(* IEC 61131-3 sources: Idecon_CheckWeigher_WP/plc_export, 11 files *)

(* ---- Idecon_BatchStats.st ---- *)
// ============================================================================
// DataType: Idecon_BatchStats
// Description: Statistiche batch da messaggio STATP (50 campi)
// Version: 1.0
// ============================================================================

TYPE Idecon_BatchStats :
STRUCT
    // === Header (Campi 1-7) ==================================================
    Timestamp               : STRING[32];       // Data/ora statistiche
    BatchStartTime          : STRING[32];       // Inizio batch
    ProductionOrder         : STRING[64];       // Ordine produzione
    ProductionCode          : STRING[64];       // Codice prodotto
    RecipeName              : STRING[32];       // Nome ricetta
    LineCode                : STRING[32];       // Codice linea
    SerialNumber            : STRING[16];       // Serial number

    // === Contatori Global Batch (Campi 8-22) =================================
    TotalProducts           : UDINT;            // Totale pezzi (Campo 8)
    TotalAccepted           : UDINT;            // Totale accettati (Campo 9)
    RejectedMinusMinus      : UDINT;            // Scartati -- (Campo 13)
    RejectedMinus           : UDINT;            // Scartati - (Campo 14)
    RejectedPlus            : UDINT;            // Scartati + (Campo 15)
    RejectedPlusPlus        : UDINT;            // Scartati ++ (Campo 16)
    CannotBeWeighed         : UDINT;            // Non pesabili (Campo 17)
    MetalDetected           : UDINT;            // Metallo rilevato (Campo 18)

    // === Metal Test (Campi 19-22) ============================================
    MetalTestsPerformed     : UDINT;            // Test metallo eseguiti
    MetalTestsPassed        : UDINT;            // Test superati
    MetalTestsFailed        : UDINT;            // Test falliti
    MetalTestsRefused       : UDINT;            // Test rifiutati

    // === Pesi Campione OK (Campi 10-12, 23-26) ===============================
    AverageWeight_g         : REAL;             // Peso medio accettati (g)
    MinWeight_g             : REAL;             // Peso minimo accettati (g)
    MaxWeight_g             : REAL;             // Peso massimo accettati (g)

    // Ultimo peso (Campi 23-26)
    LastWeightExact_g       : REAL;             // Ultimo peso esatto (g)
    LastWeightRounded_g     : REAL;             // Ultimo peso arrotondato (g)
    LastWeightDiff_g        : REAL;             // Ultimo delta (g)
    LastWeightClass         : STRING[16];       // Classe ultimo peso

    // === Contatori Incrementali (Campi 27-46) ================================
    IncrProducts            : UDINT;            // Incrementale totale
    IncrAccepted            : UDINT;            // Incrementale accettati
    IncrRejectedMM          : UDINT;            // Incrementale --
    IncrRejectedM           : UDINT;            // Incrementale -
    IncrRejectedP           : UDINT;            // Incrementale +
    IncrRejectedPP          : UDINT;            // Incrementale ++
    IncrCannotBeWeighed     : UDINT;            // Incrementale non pesabili
    IncrMetalDetected       : UDINT;            // Incrementale metallo

    // === KPI (Campi 47-50) ===================================================
    OKMinusProducts         : UDINT;            // OK- prodotti (Campo 48)
    OKMinusAccepted         : UDINT;            // OK- accettati (Campo 49)
    StandardDeviation_g     : REAL;             // Deviazione standard (Campo 50)

    // === KPI Calcolati =======================================================
    YieldPercentage         : REAL;             // Rendimento % (Accepted/Total*100)
    RejectionRate           : REAL;             // Tasso scarto %
    ProductionRate_PPM      : REAL;             // Pezzi al minuto
    TotalWeight_kg          : REAL;             // Peso totale kg

    // === Stato e Validità ====================================================
    BatchActive             : BOOL;             // Batch attivo
    DataValid               : BOOL;             // Dati validi
    ReceivedTime            : LINT;             // Timestamp ricezione
    LastUpdateTime          : LINT;             // Ultimo aggiornamento
    ParseError              : BOOL;             // Errore parsing
    ErrorCode               : UINT;             // Codice errore

    // === Campi Extra dal Batch ===============================================
    ExtraField1             : STRING[64];       // Campo extra 1
    ExtraField2             : STRING[64];       // Campo extra 2
    UserName                : STRING[32];       // Nome operatore

END_STRUCT;
END_TYPE

(* ---- Idecon_Command.st ---- *)
// ============================================================================
// DataType: Idecon_Command
// Description: Struttura per gestione comando singolo verso bilancia
// ============================================================================

TYPE Idecon_Command :
STRUCT
    // === Input (da programma chiamante) ======================================
    Execute                 : BOOL;             // Esegui comando (fronte salita)
    Command                 : STRING[255];      // Stringa comando (es. "STATSV")
    Timeout                 : TIME := T#5S;     // Timeout attesa risposta

    // === Output (da FB_IDECON_Client) ========================================
    Done                    : BOOL;             // Comando completato con successo
    Busy                    : BOOL;             // Comando in esecuzione
    Error                   : BOOL;             // Errore durante esecuzione
    ErrorID                 : WORD;             // Codice errore specifico

    // === Risposta ============================================================
    Response                : STRING[512];      // Risposta testuale da bilancia
    ResponseRaw             : ARRAY[0..511] OF BYTE;  // Risposta come array byte
    ResponseLen             : UINT;             // Lunghezza risposta in bytes
    ResponseTime_ms         : UDINT;            // Tempo risposta (ms)

    // === Timestamp ===========================================================
    ExecuteTime             : LINT;             // Quando è stato eseguito
    DoneTime                : LINT;             // Quando è stato completato

END_STRUCT;
END_TYPE

(* ---- Idecon_CommStatus.st ---- *)
// ============================================================================
// DataType: Idecon_CommStatus
// Description: Stato comunicazione TCP con bilancia IDECON
// ============================================================================

TYPE Idecon_CommStatus :
STRUCT
    // === Stato Connessione ===================================================
    Connected               : BOOL;             // Socket connesso fisicamente
    Online                  : BOOL;             // Comunicazione attiva (ultimo msg < timeout)
    Ready                   : BOOL;             // Pronto per inviare comandi

    // === Statistiche Comunicazione ===========================================
    RxCount                 : UDINT;            // Totale messaggi ricevuti
    TxCount                 : UDINT;            // Totale comandi inviati
    ErrorCount              : UDINT;            // Contatore errori
    RetryCount              : UINT;             // Retry in corso

    // === Timestamp ===========================================================
    LastRxTime              : LINT;             // Timestamp ultimo messaggio ricevuto (Unix ms)
    LastTxTime              : LINT;             // Timestamp ultimo comando inviato
    ConnectionTime          : LINT;             // Timestamp connessione stabilita

    // === Errori ==============================================================
    LastError               : WORD;             // Codice ultimo errore
    LastErrorTime           : LINT;             // Timestamp ultimo errore

    // === Stato Dettagliato ===================================================
    StatusCode              : STRING[8];        // Ultimo STATSV ricevuto
    WorkMode                : UINT;             // 1=LOCAL, 2=REMOTE, 3=MAINTENANCE
    IsLocalMode             : BOOL;             // TRUE se in LOCAL
    IsRemoteMode            : BOOL;             // TRUE se in REMOTE

END_STRUCT;
END_TYPE

(* ---- Idecon_Config.st ---- *)
// ============================================================================
// DataType: Ideon_Config
// Description: Configurazione rete e parametri bilancia IDECON
// ============================================================================

TYPE Idecon_Config :
STRUCT
    // === Parametri Rete ======================================================
    IpAddress               : STRING[15] := '172.16.224.210';  // IP bilancia
    TcpPort                 : UINT := 50000;                    // Porta TCP

    // === Timeout (millisecondi) ==============================================
    ConnectionTimeout_ms    : UDINT := 10000;                   // Timeout connessione
    CommandTimeout_ms       : UDINT := 5000;                    // Timeout comando
    ResponseTimeout_ms      : UDINT := 5000;                    // Timeout risposta

    // === Polling =============================================================
    PollInterval_ms         : UDINT := 5000;                    // Intervallo polling STATSV

    // === Retry ===============================================================
    MaxRetries              : UINT := 3;                        // Numero max retry

    // === MSGFILTER ===========================================================
    MsgFilterValue          : UINT := 23;                       // 0b10111 = risp+err+ev+pesi

    // === Statistiche =========================================================
    StatsCadency_sec        : UINT := 30;                       // Frequenza STATP (secondi)

    // === Abilitazione ========================================================
    Connect                 : BOOL := FALSE;                    // Abilita connessione
    AutoReconnect           : BOOL := TRUE;                     // Riconnessione automatica

END_STRUCT;
END_TYPE

(* ---- Idecon_LocalStats.st ---- *)
// ============================================================================
// DataType: Idecon_LocalStats
// Description: Statistiche locali calcolate dal PLC (indipendenti da bilancia)
// ============================================================================

TYPE Idecon_LocalStats :
STRUCT
    // === Contatori Totali ====================================================
    TotalWeights            : UDINT;            // Totale pesi ricevuti
    TotalAccepted           : UDINT;            // Totale OK
    TotalRejected           : UDINT;            // Totale scartati
    TotalExpelled           : UDINT;            // Totale espulsi

    // === Contatori per Categoria =============================================
    CountOK                 : UDINT;            // Solo OK
    CountOKPlus             : UDINT;            // OK+
    CountOKMinus            : UDINT;            // OK-
    CountPlus               : UDINT;            // +
    CountPlusPlus           : UDINT;            // ++
    CountMinus              : UDINT;            // -
    CountMinusMinus         : UDINT;            // --
    CountMetal              : UDINT;            // Con metallo

    // === Pesi (calcolati in g) ===============================================
    SumWeight_g             : REAL;             // Somma pesi (per media)
    AvgWeight_g             : REAL;             // Media pesi
    MinWeight_g             : REAL;             // Peso minimo rilevato
    MaxWeight_g             : REAL;             // Peso massimo rilevato

    // === Timing ==============================================================
    FirstWeightTime         : LINT;             // Timestamp prima pesata
    LastWeightTime          : LINT;            // Timestamp ultima pesata
    ProductionTime_sec      : UDINT;            // Tempo produzione (secondi)

    // === Allarmi =============================================================
    Error30_Count           : UDINT;            // Quanti errori 30 ricevuti
    OtherErrors_Count       : UDINT;            // Altri errori

    // === Reset ===============================================================
    Reset                   : BOOL;             // Azzera contatori

END_STRUCT;
END_TYPE

(* ---- Idecon_Types.st ---- *)
// ============================================================================
// DataType: Idecon_Status
// Description: Stato macchina da risposta STATSV
// Version: 1.0
// ============================================================================

TYPE Idecon_Status :
STRUCT
    // === Codice Stato (8 caratteri) ==========================================
    StatusCode              : STRING[8];        // Codice completo (es. "20110011")

    // === Posizione 1: Stato Motori ==========================================
    MotorStatus             : UINT;             // 0=Fermo, 1=Regolazione, 2=Pronto, 3=Standby, 4=Ripresa
    MotorRunning            : BOOL;             // TRUE se in moto

    // === Posizione 2: Produzione =============================================
    ProductionStarted       : BOOL;             // 1=Produzione attiva

    // === Posizione 3-5: Allarmi ==============================================
    HasErrors               : BOOL;             // 1=Errori presenti
    HasWarnings             : BOOL;             // 1=Warning presenti
    HasMessages             : BOOL;             // 1=Messaggi presenti

    // === Posizione 6: Statistiche ============================================
    StatsEnabled            : BOOL;             // 1=Invio STATP abilitato

    // === Posizione 7: Modalità Operativa =====================================
    WorkMode                : UINT;             // 1=LOCAL, 2=REMOTE, 3=MAINTENANCE
    IsLocalMode             : BOOL;             // TRUE se in LOCAL
    IsRemoteMode            : BOOL;             // TRUE se in REMOTE
    IsMaintenanceMode       : BOOL;             // TRUE se in MAINTENANCE

    // === Posizione 8: Connessione ============================================
    ConnectionStatus        : UINT;             // Stato connessione

    // === Timestamp ===========================================================
    ReceivedTime            : LINT;             // Timestamp ricezione
    Valid                   : BOOL;             // Dati validi

END_STRUCT;
END_TYPE

// ============================================================================
// DataType: Idecon_EventData
// Description: Dati evento da messaggio EVENT
// Version: 1.0
// ============================================================================

TYPE Idecon_EventData :
STRUCT
    Timestamp               : STRING[32];       // Data/ora evento
    ProductionOrder         : STRING[64];       // Ordine
    BatchCode               : STRING[64];       // Batch
    RecipeName              : STRING[32];       // Ricetta
    LineCode                : STRING[32];       // Linea
    SerialNumber            : STRING[16];       // Serial

    EventCode               : UINT;             // Codice evento (1000-9999)
    EventDescription        : STRING[255];      // Descrizione testuale
    Operator                : STRING[32];       // Operatore

    // Flag comuni
    IsError                 : BOOL;             // TRUE se errore
    IsWarning               : BOOL;             // TRUE se warning
    IsInfo                  : BOOL;             // TRUE se informativo

    // Timestamp
    ReceivedTime            : LINT;
    Valid                   : BOOL;

END_STRUCT;
END_TYPE

// ============================================================================
// DataType: Idecon_Config
// Description: Configurazione connessione IDECON
// Version: 1.0
// ============================================================================

TYPE Idecon_Config :
STRUCT
    // === Parametri Rete ======================================================
    IpAddress               : STRING[15];       // IP bilancia (es. "172.16.224.210")
    TcpPort                 : UINT;             // Porta (default 50000)

    // === Timeout =============================================================
    ConnectionTimeout_ms    : UDINT;            // Timeout connessione (ms)
    CommandTimeout_ms       : UDINT;            // Timeout comando (ms)
    ResponseTimeout_ms      : UDINT;            // Timeout risposta (ms)

    // === Polling =============================================================
    PollInterval_ms         : UDINT;            // Intervallo polling STATSV (ms)

    // === Retry ===============================================================
    MaxRetries              : UINT;             // Numero massimo retry

    // === MSGFILTER ===========================================================
    MsgFilterValue          : UINT;             // Valore MSGFILTER (default 23)

    // === Statistiche =========================================================
    StatsCadency_sec        : UINT;             // Frequenza STATP (default 30s)

    // === Abilitazione ========================================================
    Connect                 : BOOL;             // Abilita connessione
    AutoReconnect           : BOOL;             // Riconnessione automatica

END_STRUCT;
END_TYPE

(* ---- Idecon_WeightData.st ---- *)
// ============================================================================
// DataType: Idecon_WeightData
// Description: Struttura dati per messaggio WEIGHT dalla bilancia IDECON
// Version: 1.0
// ============================================================================

TYPE Idecon_WeightData :
STRUCT
    // === Identificazione =====================================================
    Timestamp               : STRING[32];       // Data/ora pesata (yyyy.mm.dd hh:mm:ss:msec)
    ProductionOrder         : STRING[64];       // Ordine produzione
    BatchCode               : STRING[64];       // Codice batch/lotto
    RecipeName              : STRING[32];       // Nome ricetta (es. "225g")
    LineCode                : STRING[32];       // Codice linea
    SerialNumber            : STRING[16];       // Serial number bilancia

    // === Valori numerici (in milligrammi) ====================================
    WeightMg                : DINT;             // Peso rilevato in mg
    DeltaMg                 : DINT;             // Delta da peso nominale in mg
    Classification          : UDINT;            // Bitmap classificazione (19 bit)

    // === Flag decodificati (19 bit di Classification) ========================
    // Bit 0-2: Caratteristiche fisiche
    FlagProductTooLong      : BOOL;             // Prodotto troppo lungo (Bit 0)
    FlagProductTooShort     : BOOL;             // Prodotto troppo corto (Bit 1)
    FlagMetal               : BOOL;             // Rilevato metallo (Bit 2)

    // Bit 3-7: Categorie peso
    FlagWeightPlusPlus      : BOOL;             // Categoria ++ (Bit 3)
    FlagWeightPlus          : BOOL;             // Categoria + (Bit 4)
    FlagWeightMinusMinus    : BOOL;             // Categoria -- (Bit 5)
    FlagWeightMinus         : BOOL;             // Categoria - (Bit 6)
    FlagWeightOK            : BOOL;             // Categoria OK (Bit 7)

    // Bit 8-11: Condizioni speciali
    FlagExpelled            : BOOL;             // Espulso (Bit 8)
    FlagProductTooClose     : BOOL;             // Prodotto troppo vicino (Bit 9)
    FlagNewDynamicTare      : BOOL;             // Nuova tara dinamica (Bit 10)
    FlagIncorrectTare       : BOOL;             // Tara incorretta (Bit 11)

    // Bit 12-13: Fuori range
    FlagAboveMaxCapacity    : BOOL;             // Sopra capacità max (Bit 12)
    FlagBelowMinCapacity    : BOOL;             // Sotto capacità min (Bit 13)

    // Bit 14-18: Condizioni OK speciali
    FlagOKMinusAccepted     : BOOL;             // OK- accettato (Bit 14)
    FlagNoUpstreamConsent   : BOOL;             // No consenso upstream (Bit 15)
    FlagInvalidPreweight    : BOOL;             // Peso pre-pesata invalido (Bit 16)
    FlagOKAboveNominal      : BOOL;             // OK sopra nominale (Bit 17)
    FlagOKBelowNominal      : BOOL;             // OK sotto nominale (Bit 18)

    // === Validità e timestamp ================================================
    Valid                   : BOOL;             // Dati validi (ricevuti e parsati)
    ReceivedTime            : LINT;             // Timestamp ricezione (Unix ms)
    ParseError              : BOOL;             // Errore parsing
    ErrorCode               : UINT;             // Codice errore parsing

END_STRUCT;
END_TYPE

(* ---- IdeconInterface.st ---- *)
// ============================================================================
// DataType: IdeconInterface
// Description: Struttura principale unificata per gestione bilancia IDECON
//              Unica variabile in Global Variables: G_Idecon : IdeconInterface
// Version: 1.0
// ============================================================================

TYPE IdeconInterface :
STRUCT
    // === CONFIGURAZIONE (inizializzata in HSM_SpecificationsSetting) ========
    // Esempio: G_Idecon.Config.IpAddress := '172.16.224.210';
    Config                  : Idecon_Config;

    // === SOCKET TCP (gestito da FB_IDECON_Client) ===========================
    // Non modificare direttamente, usare FB
    Socket                  : _sSOCKET;

    // === STATO COMUNICAZIONE =================================================
    // Monitoraggio stato connessione e online/offline
    Comm                    : Idecon_CommStatus;

    // === DATI RICEVUTI DALLA BILANCIA ========================================
    // Ultimi dati aggiornati automaticamente
    LastWeight              : Idecon_WeightData;    // Ultima pesata WEIGHT
    BatchStats              : Idecon_BatchStats;    // Statistiche STATP
    Status                  : Idecon_Status;        // Stato macchina STATSV
    LastEvent               : Idecon_EventData;     // Ultimo evento EVENT

    // === COMANDO ATTIVO ======================================================
    // Per inviare comandi alla bilancia
    Cmd                     : Idecon_Command;

    // === STATISTICHE LOCALI PLC ==============================================
    // Contatori e calcoli fatti dal PLC
    Stats                   : Idecon_LocalStats;

    // === FLAG ERRORE SISTEMA =================================================
    // TRUE quando c'è errore grave comunicazione
    SystemError             : BOOL;

    // === VERSIONE E DIAGNOSTICA ==============================================
    Version                 : UINT := 100;          // Versione struct (1.00)

END_STRUCT;
END_TYPE

(* ---- IDECON_Utils.st ---- *)
// ============================================================================
// Function: IDECON_StartsWith
// Description: Verifica se una stringa inizia con un prefisso
// ============================================================================

FUNCTION IDECON_StartsWith : BOOL
VAR_INPUT
    Str                     : STRING[512];      // Stringa da verificare
    Prefix                  : STRING[64];       // Prefisso da cercare
END_VAR

VAR
    StrLen                  : UINT;
    PrefixLen               : UINT;
END_VAR;

StrLen := LEN(Str);
PrefixLen := LEN(Prefix);

IF PrefixLen = 0 THEN
    IDECON_StartsWith := TRUE;
    RETURN;
END_IF;

IF StrLen < PrefixLen THEN
    IDECON_StartsWith := FALSE;
    RETURN;
END_IF;

IDECON_StartsWith := (LEFT(Str, PrefixLen) = Prefix);

END_FUNCTION

// ============================================================================
// Function: IDECON_FieldAt
// Description: Estrae campo N da stringa delimitata
// ============================================================================

FUNCTION IDECON_FieldAt : STRING[64]
VAR_INPUT
    Str                     : STRING[512];      // Stringa sorgente
    FieldNum                : UINT;             // Numero campo (1-based)
    Delimiter               : STRING[1];        // Delimitatore
END_VAR

VAR
    i                       : INT;
    CurrentField            : UINT;
    StartPos                : INT;
    StrLen                  : UINT;
END_VAR;

StrLen := LEN(Str);
IF StrLen = 0 OR FieldNum = 0 THEN
    IDECON_FieldAt := '';
    RETURN;
END_IF;

CurrentField := 1;
StartPos := 1;

FOR i := 1 TO INT#(StrLen) DO
    IF MID(Str, 1, UINT#(i)) = Delimiter THEN
        IF CurrentField = FieldNum THEN
            // Campo trovato
            IDECON_FieldAt := MID(Str, UINT#(i - StartPos), UINT#(StartPos));
            RETURN;
        END_IF;
        CurrentField := CurrentField + 1;
        StartPos := i + 1;
    END_IF;
END_FOR;

// Ultimo campo
IF CurrentField = FieldNum THEN
    IDECON_FieldAt := MID(Str, UINT#(StrLen - StartPos + 1), UINT#(StartPos));
ELSE
    IDECON_FieldAt := '';
END_IF;

END_FUNCTION

// ============================================================================
// Function: IDECON_ParseHexDword
// Description: Converte stringa esadecimale in UDINT
// ============================================================================

FUNCTION IDECON_ParseHexDword : UDINT
VAR_INPUT
    HexStr                  : STRING[16];       // Stringa hex (es. "20480")
END_VAR

VAR
    Result                  : UDINT;
    i                       : INT;
    StrLen                  : UINT;
    Digit                   : BYTE;
    CharVal                 : UDINT;
END_VAR;

StrLen := LEN(HexStr);
Result := UDINT#0;

FOR i := 1 TO INT#(StrLen) DO
    Digit := STRING_TO_BYTE(MID(HexStr, 1, UINT#(i)));

    IF Digit >= BYTE#48 AND Digit <= BYTE#57 THEN
        // '0'-'9'
        CharVal := BYTE_TO_UDINT(Digit) - UDINT#48;
    ELSIF Digit >= BYTE#65 AND Digit <= BYTE#70 THEN
        // 'A'-'F'
        CharVal := BYTE_TO_UDINT(Digit) - UDINT#55;
    ELSIF Digit >= BYTE#97 AND Digit <= BYTE#102 THEN
        // 'a'-'f'
        CharVal := BYTE_TO_UDINT(Digit) - UDINT#87;
    ELSE
        CONTINUE; // Carattere non valido, salta
    END_IF;

    Result := Result * UDINT#16 + CharVal;
END_FOR;

IDECON_ParseHexDword := Result;

END_FUNCTION

(* ---- FB_IDECON_Client.st ---- *)
// ============================================================================
// Function Block: FB_IDECON_Client
// Description: Client TCP per comunicazione con bilancia IDECON
// Version: 1.0
// ============================================================================

FUNCTION_BLOCK FB_IDECON_Client
VAR_INPUT
    Execute                 : BOOL;             // Esegui comando
    Command                 : STRING[255];      // Comando da inviare
    Timeout                 : TIME := T#5S;     // Timeout risposta
END_VAR

VAR_OUTPUT
    Done                    : BOOL;             // Comando completato con successo
    Busy                    : BOOL;             // In esecuzione
    Error                   : BOOL;             // Errore
    ErrorID                 : WORD;             // Codice errore (0=nessuno)
    Response                : STRING[512];      // Risposta ricevuta
    ResponseRaw             : ARRAY[0..511] OF BYTE; // Risposta raw bytes
    ResponseLen             : UINT;             // Lunghezza risposta
END_VAR

VAR_IN_OUT
    Socket                  : _sSOCKET;         // Socket TCP
END_VAR

VAR
    // Stato FSM
    State                   : INT := 0;         // Stato macchina

    // Timer
    TimeoutTimer            : TON;              // Timer timeout
    RetryTimer              : TON;              // Timer retry

    // Buffer
    SendBuffer              : ARRAY[0..511] OF BYTE;
    RecvBuffer              : ARRAY[0..1023] OF BYTE;
    CmdLen                  : UINT;
    RetryCount              : INT := 0;
    MaxRetries              : INT := 3;

    // Costanti protocollo
    STX                     : BYTE := BYTE#16#02;  // Start of Text
    ETX                     : BYTE := BYTE#16#03;  // End of Text

    // Variabili interne
    i                       : INT;
    j                       : INT;
    StrLen                  : UINT;
    RecvDone                : BOOL;
    SendDone                : BOOL;

END_VAR

// Stati FSM
// 0: Idle
// 1: Prepara comando
// 2: Invia STX
// 3: Invia comando
// 4: Invia ETX
// 5: Attendi risposta
// 6: Ricevi dati
// 7: Parsa risposta
// 8: Completato
// 9: Errore

// ============================================================================
// IMPLEMENTAZIONE
// ============================================================================

IF NOT Execute AND State <> 0 THEN
    // Reset su fronte negativo Execute
    State := 0;
    Busy := FALSE;
END_IF;

CASE State OF

    0: // Idle
        Done := FALSE;
        Error := FALSE;
        ErrorID := WORD#0;
        Busy := FALSE;
        RetryCount := 0;

        IF Execute THEN
            State := 1;
            Busy := TRUE;
        END_IF;

    1: // Prepara comando
        // Prepara buffer: STX + Comando + ETX
        StrLen := LEN(Command);

        IF StrLen = 0 OR StrLen > 250 THEN
            Error := TRUE;
            ErrorID := WORD#1; // Comando vuoto o troppo lungo
            State := 9;
        ELSE
            // Copia comando in buffer
            FOR i := 0 TO INT#(StrLen - 1) DO
                SendBuffer[i + 1] := STRING_TO_BYTE(MID(Command, 1, UINT#(i + 1)));
            END_FOR;

            CmdLen := StrLen;
            State := 2;
        END_IF;

    2: // Invia STX
        Socket.Send(ADR(STX), 1);

        IF Socket.Done THEN
            State := 3;
        ELSIF Socket.Error THEN
            Error := TRUE;
            ErrorID := Socket.ErrorID;
            State := 9;
        END_IF;

    3: // Invia comando
        Socket.Send(ADR(SendBuffer[1]), CmdLen);

        IF Socket.Done THEN
            State := 4;
        ELSIF Socket.Error THEN
            Error := TRUE;
            ErrorID := Socket.ErrorID;
            State := 9;
        END_IF;

    4: // Invia ETX
        Socket.Send(ADR(ETX), 1);

        IF Socket.Done THEN
            State := 5;
            TimeoutTimer(IN := TRUE, PT := Timeout);
        ELSIF Socket.Error THEN
            Error := TRUE;
            ErrorID := Socket.ErrorID;
            State := 9;
        END_IF;

    5: // Attendi risposta
        TimeoutTimer(IN := TRUE);

        IF TimeoutTimer.Q THEN
            // Timeout - retry?
            IF RetryCount < MaxRetries THEN
                RetryCount := RetryCount + 1;
                State := 1; // Riprova
                TimeoutTimer(IN := FALSE);
            ELSE
                Error := TRUE;
                ErrorID := WORD#16#8001; // Timeout
                State := 9;
            END_IF;
        END_IF;

        // Controlla se ci sono dati
        IF Socket.Available > 0 THEN
            State := 6;
            TimeoutTimer(IN := FALSE);
        END_IF;

    6: // Ricevi dati
        Socket.Recv(ADR(RecvBuffer), SIZEOF(RecvBuffer), RecvLen);

        IF Socket.Done THEN
            State := 7;
        ELSIF Socket.Error THEN
            Error := TRUE;
            ErrorID := Socket.ErrorID;
            State := 9;
        END_IF;

    7: // Parsa risposta
        // Rimuovi STX e ETX se presenti
        IF RecvLen > 0 THEN
            j := 0;
            FOR i := 0 TO INT#(RecvLen - 1) DO
                // Salta STX iniziale
                IF i = 0 AND RecvBuffer[i] = STX THEN
                    CONTINUE;
                END_IF;
                // Salta ETX finale
                IF i = INT#(RecvLen - 1) AND RecvBuffer[i] = ETX THEN
                    CONTINUE;
                END_IF;
                // Copia byte valido
                ResponseRaw[j] := RecvBuffer[i];
                j := j + 1;
            END_FOR;

            // Converti in stringa
            Response := '';
            FOR i := 0 TO j - 1 DO
                IF ResponseRaw[i] >= BYTE#32 AND ResponseRaw[i] <= BYTE#126 THEN
                    Response := CONCAT(Response, BYTE_TO_STRING(ResponseRaw[i]));
                END_IF;
            END_FOR;

            ResponseLen := UINT#(j);
        END_IF;

        State := 8;

    8: // Completato
        Done := TRUE;
        Busy := FALSE;
        Error := FALSE;

        IF NOT Execute THEN
            State := 0;
        END_IF;

    9: // Errore
        Error := TRUE;
        Busy := FALSE;
        Done := FALSE;

        IF NOT Execute THEN
            State := 0;
        END_IF;

END_CASE;

END_FUNCTION_BLOCK

(* ---- FB_ParseWeightMessage.st ---- *)
// ============================================================================
// Function Block: FB_ParseWeightMessage
// Description: Parsa messaggio WEIGHT dalla bilancia IDECON
// Version: 1.0
// ============================================================================

FUNCTION_BLOCK FB_ParseWeightMessage
VAR_INPUT
    Enable                  : BOOL;             // Abilita parsing
    Message                 : STRING[512];      // Messaggio da parsare
    MessageRaw              : ARRAY[0..511] OF BYTE;
    MessageLen              : UINT;
END_VAR

VAR_OUTPUT
    Done                    : BOOL;             // Parsing completato
    Error                   : BOOL;             // Errore parsing
    ErrorCode               : UINT;             // Codice errore
    WeightData              : Idecon_WeightData; // Dati peso parsati
END_VAR

VAR
    // Variabili interne
    MsgTemp                 : STRING[512];
    Parts                   : ARRAY[0..10] OF STRING[64];
    NumParts                : INT;
    i                       : INT;
    Pos                     : INT;
    LastPos                 : INT;
    ClassificationValue     : UDINT;

END_VAR

// ============================================================================
// IMPLEMENTAZIONE
// ============================================================================

IF NOT Enable THEN
    Done := FALSE;
    Error := FALSE;
    ErrorCode := UINT#0;
    RETURN;
END_IF;

// Verifica prefisso WEIGHT=
IF NOT IDECON_StartsWith(Message, 'WEIGHT=') THEN
    Error := TRUE;
    ErrorCode := UINT#1; // Prefisso non valido
    RETURN;
END_IF;

// Rimuovi prefisso
MsgTemp := DELETE(Message, 7, 1); // Rimuovi "WEIGHT="

// Split per |
NumParts := 0;
Pos := 1;
LastPos := 1;

FOR i := 1 TO LEN(MsgTemp) DO
    IF MID(MsgTemp, 1, UINT#(i)) = '|' THEN
        IF NumParts <= 9 THEN
            Parts[NumParts] := MID(MsgTemp, UINT#(i - LastPos), UINT#(LastPos));
            NumParts := NumParts + 1;
            LastPos := i + 1;
        END_IF;
    END_IF;
END_FOR;

// Ultimo campo
IF NumParts <= 9 AND LastPos <= LEN(MsgTemp) THEN
    Parts[NumParts] := MID(MsgTemp, UINT#(LEN(MsgTemp) - LastPos + 1), UINT#(LastPos));
    NumParts := NumParts + 1;
END_IF;

// Verifica numero campi
IF NumParts < 9 THEN
    Error := TRUE;
    ErrorCode := UINT#2; // Numero campi insufficiente
    WeightData.ParseError := TRUE;
    WeightData.ErrorCode := UINT#2;
    RETURN;
END_IF;

// Parsing campi
WeightData.Timestamp := Parts[0];
WeightData.ProductionOrder := Parts[1];
WeightData.BatchCode := Parts[2];
WeightData.RecipeName := Parts[3];
WeightData.LineCode := Parts[4];
WeightData.SerialNumber := Parts[5];

// Conversione numerica
WeightData.WeightMg := STRING_TO_DINT(Parts[6]);
WeightData.DeltaMg := STRING_TO_DINT(Parts[7]);

// Parsing classification (hex)
ClassificationValue := STRING_TO_UDINT(Parts[8]);
WeightData.Classification := ClassificationValue;

// Decodifica bit
WeightData.FlagProductTooLong := (ClassificationValue AND UDINT#16#000001) > UDINT#0;
WeightData.FlagProductTooShort := (ClassificationValue AND UDINT#16#000002) > UDINT#0;
WeightData.FlagMetal := (ClassificationValue AND UDINT#16#000004) > UDINT#0;
WeightData.FlagWeightPlusPlus := (ClassificationValue AND UDINT#16#000008) > UDINT#0;
WeightData.FlagWeightPlus := (ClassificationValue AND UDINT#16#000010) > UDINT#0;
WeightData.FlagWeightMinusMinus := (ClassificationValue AND UDINT#16#000020) > UDINT#0;
WeightData.FlagWeightMinus := (ClassificationValue AND UDINT#16#000040) > UDINT#0;
WeightData.FlagWeightOK := (ClassificationValue AND UDINT#16#000080) > UDINT#0;
WeightData.FlagExpelled := (ClassificationValue AND UDINT#16#000100) > UDINT#0;
WeightData.FlagProductTooClose := (ClassificationValue AND UDINT#16#000200) > UDINT#0;
WeightData.FlagNewDynamicTare := (ClassificationValue AND UDINT#16#000400) > UDINT#0;
WeightData.FlagIncorrectTare := (ClassificationValue AND UDINT#16#000800) > UDINT#0;
WeightData.FlagAboveMaxCapacity := (ClassificationValue AND UDINT#16#001000) > UDINT#0;
WeightData.FlagBelowMinCapacity := (ClassificationValue AND UDINT#16#002000) > UDINT#0;
WeightData.FlagOKMinusAccepted := (ClassificationValue AND UDINT#16#004000) > UDINT#0;
WeightData.FlagNoUpstreamConsent := (ClassificationValue AND UDINT#16#008000) > UDINT#0;
WeightData.FlagInvalidPreweight := (ClassificationValue AND UDINT#16#010000) > UDINT#0;
WeightData.FlagOKAboveNominal := (ClassificationValue AND UDINT#16#020000) > UDINT#0;
WeightData.FlagOKBelowNominal := (ClassificationValue AND UDINT#16#040000) > UDINT#0;

// Validazione
WeightData.Valid := TRUE;
WeightData.ParseError := FALSE;
WeightData.ErrorCode := UINT#0;
WeightData.ReceivedTime := 0; // Da impostare chiamante

Done := TRUE;
Error := FALSE;

END_FUNCTION_BLOCK
